Universal Robots PolyScope program: orange_Dovetail_buttom.urp

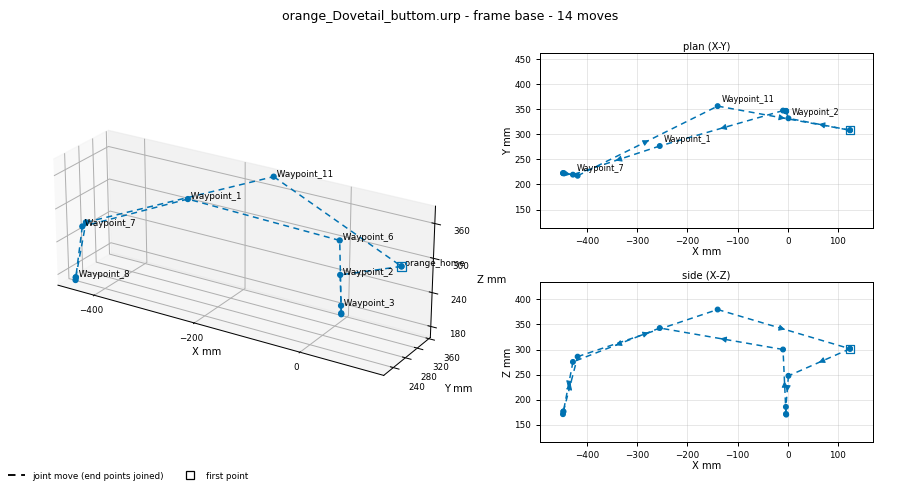
[picture p0: tool path of orange_Dovetail_buttom.urp in frame base, 14 of 14 moves have a stored position in this frame; points joined in program order, loops and branches not executed]
Program orange_Dovetail_buttom (installation=default directory=/programs/usbdisk/Zahra1/orangi createdIn=5.11.11.1010533 lastSavedIn=5.11.11.1010533 robotSerialNumber=20205300864)
Calibrated DH parameters: a=[-0.000166, -0.243494, -0.153108, 0.000057, -0.000123, 0]; d=[0.151897, -1.34267, 53.988124, -52.514559, 0.085283, 0.092193]; alpha=[1.572472, -0.003756, 0.002824, 1.570807, -1.572621, 0]; deltaTheta=[0, 0.020704, 7.033215, -0.770746, 0.000004, 0]
Robot Program (runOnlyOnce=true)
  MoveJ speed 60 deg/s, acceleration 80 deg/s^2 (useActiveTCP=true) feature=Base
    Waypoint orange_home: TCP in base x=124.286 y=308.277 z=301.462 mm, rx=2.2499 ry=-2.1846 rz=-0.0963 rad; joints [-269.66, -91.226, -90.279, -86.086, 92.69, 808.818] deg
    URCap Gripper (Robotiq_Grippers, Robotiq Inc.) dataModel(position=40.3921568627451, force=97.0, speed=52.0, positionInDouble=40.3921568627451, forceInDouble=97.0, speedInDouble=52.0, slaveIds=[9], blocking=true, robotCompliant=false)
    Waypoint Waypoint_2: TCP in base x=1.402 y=331.981 z=247.481 mm, rx=-2.1655 ry=2.1658 rz=0.1293 rad; joints [-246.442, -91.401, -106.515, -65.89, 87.74, 833.589] deg
    Waypoint Waypoint_3: TCP in base x=-3.639 y=346.03 z=185.549 mm, rx=-2.1922 ry=2.199 rz=-0.0374 rad; joints [-246.598, -102.421, -109.091, -58.912, 87.581, 833.762] deg
    Waypoint Waypoint_4: TCP in base x=-2.97 y=346.158 z=170.1 mm, rx=-2.1922 ry=2.199 rz=-0.0375 rad; joints [-246.722, -104.59, -111.209, -54.623, 87.572, 833.651] deg
    URCap Gripper (Robotiq_Grippers, Robotiq Inc.) dataModel(position=76.58823529411765, force=97.0, speed=52.0, positionInDouble=76.58823529411765, forceInDouble=97.0, speedInDouble=52.0, slaveIds=[9], blocking=true, robotCompliant=false)
    Waypoint Waypoint_5: TCP in base x=-3.501 y=346.946 z=171.514 mm, rx=-2.1967 ry=2.2032 rz=-0.0544 rad; joints [-246.722, -104.661, -110.302, -56.169, 87.686, 833.652] deg
    Waypoint Waypoint_6: TCP in base x=-9.383 y=347.429 z=300.038 mm, rx=-2.1967 ry=2.2032 rz=-0.0543 rad; joints [-245.751, -95.633, -84.49, -91.042, 87.698, 834.543] deg
    Waypoint Waypoint_1: TCP in base x=-255.281 y=276.773 z=342.85 mm, rx=-2.3788 ry=1.9995 rz=0.1145 rad; joints [-206.295, -102.005, -67.446, -96.781, 87.172, 863.785] deg
    Waypoint Waypoint_7: TCP in base x=-428.484 y=219.609 z=275.271 mm, rx=2.1086 ry=-2.2589 rz=-0.1128 rad; joints [-191.358, -130.491, -43.437, -90.921, 89.734, 892.61] deg
    Waypoint Waypoint_8: TCP in base x=-447.532 y=222.447 z=176.281 mm, rx=-2.1773 ry=2.2235 rz=-0.0787 rad; joints [-191.344, -141.795, -46.065, -85.351, 90.148, 889.899] deg
    Waypoint Waypoint_9: TCP in base x=-448.375 y=222.635 z=170.964 mm, rx=-2.1753 ry=2.2213 rz=-0.0851 rad; joints [-191.348, -142.464, -46.12, -84.914, 90.148, 889.894] deg
    URCap Gripper (Robotiq_Grippers, Robotiq Inc.) dataModel(position=38.431372549019606, force=97.0, speed=52.0, positionInDouble=38.431372549019606, forceInDouble=97.0, speedInDouble=52.0, slaveIds=[9], blocking=true, robotCompliant=false)
    Waypoint Waypoint_8: TCP in base x=-447.532 y=222.447 z=176.281 mm, rx=-2.1773 ry=2.2235 rz=-0.0787 rad; joints [-191.344, -141.795, -46.065, -85.351, 90.148, 889.899] deg
    Waypoint Waypoint_10: TCP in base x=-419.134 y=217.396 z=285.762 mm, rx=2.1691 ry=-2.2157 rz=-0.0854 rad; joints [-191.364, -128.336, -43.826, -93.845, 89.977, 889.896] deg
    Waypoint Waypoint_11: TCP in base x=-139.828 y=356.346 z=379.778 mm, rx=-1.4379 ry=2.7872 rz=-0.0305 rad; joints [-228.581, -110.289, -43.764, -116.997, 89.873, 886.894] deg
    Waypoint orange_home: TCP in base x=124.286 y=308.277 z=301.462 mm, rx=2.2499 ry=-2.1846 rz=-0.0963 rad; joints [-269.66, -91.226, -90.279, -86.086, 92.69, 808.818] deg
